FUNCTION_BLOCK E_MERGE2
  (* Version 1.0, 2005-05-11, Goran Cengic, Chalmers *)
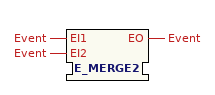
  EVENT_INPUT
    EI1;
    EI2;
  END_EVENT
  EVENT_OUTPUT
    EO;
  END_EVENT
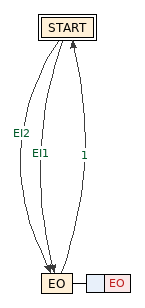
  EC_STATES
    START;
    EO : -> EO;
  END_STATES
  EC_TRANSITIONS
    START TO EO := EI1;
    START TO EO := EI2;
    EO TO START := 1;
  END_TRANSITIONS
END_FUNCTION_BLOCK
